TYPE ST_AlarmString :
STRUCT
	chinese:		STRING:='CN';
	english:		STRING:='EN';
END_STRUCT
END_TYPE

(* stored: Version 1.1.0.1, ProductVersion 3.1.4024.12
   DUT ST_AlarmString: Id {d05f9ad1-ef3b-4179-8374-024334786286} *)
